// TIA Portal V20 export
DATA_BLOCK "Alarms"   // DB149
// stored: Access Published, MemoryReserve 100, Namespace Unit1
   VAR
      unitAlarms { ExternalWritable := 'False'} : "LAF_typeAlarms";
      emAlarms { ExternalWritable := 'False'} : Array[0.._.U1_NO_OF_EMs] of "LAF_typeAlarms";
      maintenanceFaults { ExternalWritable := 'False'} : Array[0..199] of Bool;   // PFE Maintenance Faults
      productionFaults { ExternalWritable := 'False'} : Array[0..199] of Bool;   // PFE Production Faults
      toolingFault { ExternalWritable := 'False'} : Array[0..199] of Bool;   // PFE Tooling Faults
      qualityFault { ExternalWritable := 'False'} : Array[0..199] of Bool;   // PFE Quality Faults
      throughputFaultBlocked { ExternalWritable := 'False'} : Array[0..199] of Bool;   // PFE Throughput Fault Blocked
      throughputFaultStarved { ExternalWritable := 'False'} : Array[0..199] of Bool;   // PFE Throughput Fault Starved
      throughputFault { ExternalWritable := 'False'} : Array[0..199] of Bool;   // PFE Throughput Fault
      systemFaultGeneral { ExternalWritable := 'False'} : Array[0..199] of Bool;   // PFE System Fault General
      materialFault { ExternalWritable := 'False'} : Array[0..199] of Bool;   // PFE Material Fault
      maintenanceWarnings { ExternalWritable := 'False'} : Array[0..199] of Bool;   // PFE Maintenance Warnings
      productionWarning { ExternalWritable := 'False'} : Array[0..199] of Bool;   // PFE Production Warning
      toolingWarning { ExternalWritable := 'False'} : Array[0..199] of Bool;   // PFE Tooling Warning
      qualityWarning { ExternalWritable := 'False'} : Array[0..199] of Bool;   // PFE Quality Warning
      throughputWarning { ExternalWritable := 'False'} : Array[0..199] of Bool;   // PFE Throughput Warning
      systemWarning { ExternalWritable := 'False'} : Array[0..199] of Bool;   // PFE System Warning
      materialWarning { ExternalWritable := 'False'} : Array[0..199] of Bool;   // PFE Material Warning
      maintenanceStatus { ExternalWritable := 'False'} : Array[0..199] of Bool;   // PFE Maintenance Status
      productionStatus { ExternalWritable := 'False'} : Array[0..199] of Bool;   // PFE Production Status
      toolingStatus { ExternalWritable := 'False'} : Array[0..199] of Bool;   // PFE Tooling Status
      qualityStatus { ExternalWritable := 'False'} : Array[0..199] of Bool;   // PFE Quality Status
      throughputStatus { ExternalWritable := 'False'} : Array[0..199] of Bool;   // PFE Throughput Status
      systemStatus { ExternalWritable := 'False'} : Array[0..199] of Bool;   // PFE System Status
      materialStatus { ExternalWritable := 'False'} : Array[0..199] of Bool;   // PFE Material Status
      tonMaintenanceFault { ExternalWritable := 'False'} : Array[0..199] of TON_TIME;   // PFE Maintenance Faults Ton Timer
      tonProductionFault { ExternalWritable := 'False'} : Array[0..199] of TON_TIME;   // PFE Production Faults Ton Timer
      tonToolingFault { ExternalWritable := 'False'} : Array[0..199] of TON_TIME;   // PFE Tooling Faults Ton Timer
      tonQualityFault { ExternalWritable := 'False'} : Array[0..199] of TON_TIME;   // PFE Quality Faults Ton Timer
      tonThroughputFaultBlocked { ExternalWritable := 'False'} : Array[0..199] of TON_TIME;   // PFE Throughput Fault Blocked Ton Timer
      tonThroughputFaultStarved { ExternalWritable := 'False'} : Array[0..199] of TON_TIME;   // PFE Throughput Fault Starved Ton Timer
      tonThroughputFault { ExternalWritable := 'False'} : Array[0..199] of TON_TIME;   // PFE Throughput Fault Ton Timer
      tonSystemFaultGeneral { ExternalWritable := 'False'} : Array[0..199] of TON_TIME;   // PFE System Fault General Ton Timer
      tonMaterialFault { ExternalWritable := 'False'} : Array[0..199] of TON_TIME;   // PFE Material Fault Ton Timer
      tonMaintenanceWarning { ExternalWritable := 'False'} : Array[0..199] of TON_TIME;   // PFE Maintenance Warnings Ton Timer
      tonProductionWarning { ExternalWritable := 'False'} : Array[0..199] of TON_TIME;   // PFE Production Warning Ton Timer
      tonToolingWarning { ExternalWritable := 'False'} : Array[0..199] of TON_TIME;   // PFE Tooling Warning Ton Timer
      tonQualityWarning { ExternalWritable := 'False'} : Array[0..199] of TON_TIME;   // PFE Quality Warning Ton Timer
      tonThroughputWarning { ExternalWritable := 'False'} : Array[0..199] of TON_TIME;   // PFE Throughput Warning Ton Timer
      tonSystemWarning { ExternalWritable := 'False'} : Array[0..199] of TON_TIME;   // PFE System Warning Ton Timer
      tonMaterialWarning { ExternalWritable := 'False'} : Array[0..199] of TON_TIME;   // PFE Material Warning Ton Timer
      tonMaintenanceStatus { ExternalWritable := 'False'} : Array[0..199] of TON_TIME;   // PFE Maintenance Status Ton Timer
      tonProductionStatus { ExternalWritable := 'False'} : Array[0..199] of TON_TIME;   // PFE Production Status Ton Timer
      tonToolingStatus { ExternalWritable := 'False'} : Array[0..199] of TON_TIME;   // PFE Tooling Status Ton Timer
      tonQualityStatus { ExternalWritable := 'False'} : Array[0..199] of TON_TIME;   // PFE Quality Status Ton Timer
      tonThroughputStatus { ExternalWritable := 'False'} : Array[0..199] of TON_TIME;   // PFE Throughput Status Ton Timer
      tonSystemStatus { ExternalWritable := 'False'} : Array[0..199] of TON_TIME;   // PFE System Status Ton Timer
      tonMaterialStatus { ExternalWritable := 'False'} : Array[0..199] of TON_TIME;   // PFE Material Status Ton Timer
      TonTimer { ExternalWritable := 'False'} : Array[0..99] of TON_TIME;
      NoDataTransfer { S7_SetPoint := 'True'} : Array[0..20] of Bool;
   END_VAR
BEGIN
   // maintenanceFaults[10] : OUT P&P GRIPPER 1ST Y-AXIS ROBOT HOME SENSOR
   // maintenanceFaults[11] : OUT P&P GRIPPER 2ND Y-AXIS ROBOT HOME SENSOR
   // maintenanceFaults[12] : OUT P&P GRIPPER 1ST Z-AXIS HOME SENSOR
   // maintenanceFaults[13] : OUT P&P GRIPPER 2ND Z-AXIS HOME SENSOR
   // maintenanceFaults[14] : TAPE Attachment ROBOT HOMING SENSOR
   // maintenanceFaults[15] : TOP TAPE fix STAGE ROBOT HOME SENSOR
   // maintenanceFaults[16] : SIDE TAPE Attachment FORWARD/BACKWARD ROBOT HOME SENSOR
   // maintenanceFaults[17] : SIDE TAPE Attachment MOVER ROBOT HOME SENSOR
   // maintenanceFaults[18] : SIDE TAPE FIX STAGE HOMING SENSOR
   // maintenanceFaults[19] : SIDE TAPE FIX STAGE ROTATION HOMING SENSOR
   // maintenanceFaults[20] : Thickness Z-AXIS HOME SENSOR
   // maintenanceFaults[21] : Process P&P X-axis Head#1 HOMING SENSOR
   // maintenanceFaults[22] : Process P&P X-axis Head#2 HOMING SENSOR
   // maintenanceFaults[23] : Process P&P Y-axis Head#1 HOMING SENSOR
   // maintenanceFaults[24] : Process P&P Z-axis Head#1 HOMING SENSOR
   // maintenanceFaults[25] : Process P&P Y-axis Head#2 HOMING SENSOR
   // maintenanceFaults[26] : Process P&P Z-axis Head#2 HOMING SENSOR
   // maintenanceFaults[27] : Unloading P&P X-axis HOMING SENSOR
   // maintenanceFaults[28] : Unloading P&P Z-axis HOMING SENSOR
   // maintenanceFaults[29] : Unloading P&P Θ-axis HOMING SENSOR
   // maintenanceFaults[30] : Brake Test After 24 Hours
   // systemFaultGeneral[0] : E202CB : KISTLER 100KN PRESS POWER TRIPPED
   // systemFaultGeneral[1] : E208CB : KISTLER 100KN PRESS POWER TRIPPED
   // systemFaultGeneral[2] : E214CB : KISTLER 30KN PRESS POWER TRIPPED
   // systemFaultGeneral[3] : SPARE
   // systemFaultGeneral[4] : SPARE
   // systemFaultGeneral[5] : E320CB : E8404PWS CONTROLLER POWER SMPS AC POWER TRIPPED
   // systemFaultGeneral[6] : E326CB : E8704PWS SAFETY POWER SMPS AC POWER TRIPPED
   // systemFaultGeneral[7] : E332CB : E8804PWS CONTRL POWER SMPS AC POWER TRIPPED
   // systemFaultGeneral[8] : E4120CB : PROCESSOR POWER ON TIPPRED
   // systemFaultGeneral[9] : E4126CB : PROGRAMING POWER OUTLET TRPPED
   // systemFaultGeneral[10] : SPARE
   // systemFaultGeneral[11] : E4304CB : PANEL LED POWER TRIPPED
   // systemFaultGeneral[12] : SPARE
   // systemFaultGeneral[13] : E4420CB : CONTROL LEVEL HUB POWER TRIPPED
   // systemFaultGeneral[14] : E4426CB : MAIN HMI POWER TRIPPED
   // systemFaultGeneral[15] : E4432CB : PORTABLE HMI POWER TIPPED
   // systemFaultGeneral[16] : E4456CB : PORTABLE HMI POWER TIPPED
   // systemFaultGeneral[17] : E5100CB : 120VAC HEATER-1 POWER TR PRIMARY TRIPPED
   // systemFaultGeneral[18] : SPARE
   // systemFaultGeneral[19] : SPARE
   // systemFaultGeneral[20] : E5156CB : UPPER 1-1 HEATER POWER TRIPPED
   // systemFaultGeneral[21] : E5162CB : UPPER 1-2 HEATER POWER TRIPPED
   // systemFaultGeneral[22] : E5168CB : LOWER 1-1 HEATER POWER TRIPPED
   // systemFaultGeneral[23] : E5174CB : LOWER 1-2 HEATER POWER TRIPPED
   // systemFaultGeneral[24] : E5180CB : LOWER 1-3 HEATER POWER TRIPPED
   // systemFaultGeneral[25] : SPARE
   // systemFaultGeneral[26] : E6100CB : 120VAC HEATER-2 POWER TR PRIMARY TRIPPED
   // systemFaultGeneral[27] : SPARE
   // systemFaultGeneral[28] : SPARE
   // systemFaultGeneral[29] : E6156CB : UPPER 2-1 HEATER POWER TRIPPED
   // systemFaultGeneral[30] : E6162CB : UPPER 2-2 HEATER POWER TRIPPED
   // systemFaultGeneral[31] : E6168CB : LOWER 2-1 HEATER POWER TRIPPED
   // systemFaultGeneral[32] : E6174CB : LOWER 2-2 HEATER POWER TRIPPED
   // systemFaultGeneral[33] : E6180CB : LOWER 2-3 HEATER POWER TRIPPED
   // systemFaultGeneral[34] : SPARE
   // systemFaultGeneral[35] : E7100CB : 120VAC CONTROL POWER TR PRIMARY TRIPPED
   // systemFaultGeneral[36] : E7110CB : 120VAC CONTROL POWER TR SECONDARY TRIPPED
   // systemFaultGeneral[37] : E7116CB : CONTROL POWER ON TRIPPED
   // systemFaultGeneral[38] : E7154CB : MOTOR PANEL CONTROL POWER TRIPPED
   // systemFaultGeneral[39] : E7160CB : POWER STRIP OUTLET POWER TRIPPED
   // systemFaultGeneral[40] : E7166CB : POWER STRIP OUTLET POWER TRIPPED
   // systemFaultGeneral[41] : E7172CB : QR LASER MARKING TRIPPED
   // systemFaultGeneral[42] : E7178CB : HI-POT TESTER POWER TRIPPED
   // systemFaultGeneral[43] : E7222CB : FFU-1 POWER TRIPPED
   // systemFaultGeneral[44] : E5206CB : UPPER 1-1 TEMPERATURE CONTROLLER POWER TRIPPED
   // systemFaultGeneral[45] : E5212CB : UPPER 1-2 TEMPERATURE CONTROLLER POWER TRIPPED
   // systemFaultGeneral[46] : E5218CB : LOWER 1-1 TEMPERATURE CONTROLLER POWER TRIPPED
   // systemFaultGeneral[47] : E5224CB : LOWER 1-2 TEMPERATURE CONTROLLER POWER TRIPPED
   // systemFaultGeneral[48] : E5230CB : LOWER 1-3 TEMPERATURE CONTROLLER POWER TRIPPED
   // systemFaultGeneral[49] : E6206CB : UPPER 2-1 TEMPERATURE CONTROLLER POWER TRIPPED
   // systemFaultGeneral[50] : E6212CB : UPPER 2-2 TEMPERATURE CONTROLLER POWER TRIPPED
   // systemFaultGeneral[51] : E6218CB : LOWER 2-1 TEMPERATURE CONTROLLER POWER TRIPPED
   // systemFaultGeneral[52] : E6224CB : LOWER 2-2 TEMPERATURE CONTROLLER POWER TRIPPED
   // systemFaultGeneral[53] : E6230CB : LOWER 2-3 TEMPERATURE CONTROLLER POWER TRIPPED
   // systemFaultGeneral[54] : SPARE
   // systemFaultGeneral[55] : E8154CB : ET200MP I/O OUTPUT POWER TRIPPED
   // systemFaultGeneral[56] : E8180CB : JUNCTION BOX CONTROL POWER TRIPPED
   // systemFaultGeneral[57] : E8204CB : CLASS 2 SMPS POWER TRIPPED
   // systemFaultGeneral[58] : E8220CB : ET200ECO PN-1 POWER TRIPPED
   // systemFaultGeneral[59] : E8224CB : ET200ECO PN-2 POWER TRIPPED
   // systemFaultGeneral[60] : E8228CB : ET200ECO PN-3 POWER TRIPPED
   // systemFaultGeneral[61] : E8232CB : ET200ECO PN-4 POWER TRIPPED
   // systemFaultGeneral[62] : E8304CB : PANEL FAN POWER TRIPPED
   // systemFaultGeneral[63] : SPARE
   // systemFaultGeneral[64] : E8406CB : CONTROLLER DC POWER TRIPPED
   // systemFaultGeneral[65] : E8416CB : KISTLER CONTROL POWER TRIPPED
   // systemFaultGeneral[66] : E8422CB : MANIFOLD-1 POWER TRIPPED
   // systemFaultGeneral[67] : E8430CB : MANIFOLD-2 POWER TRIPPED
   // systemFaultGeneral[68] : E8456CB : QR READER POWER TRIPPED
   // systemFaultGeneral[69] : E8462CB : QR READER POWER TRIPPED
   // systemFaultGeneral[70] : E8468CB : HANDY QR READER POWER TRIPPED
   // systemFaultGeneral[71] : E8474CB : PROFINET CONVERTER POWER TRIPPED
   // systemFaultGeneral[72] : E8504CB : MONITORING RELAY POWER TRIPPED
   // systemFaultGeneral[73] : SPARE
   // systemFaultGeneral[74] : E8706CB : SAFETY DC POWER TRIPPED
   // systemFaultGeneral[75] : E8716CB : ET200SP I/O SAFETY POWER TRIPPED
   // systemFaultGeneral[76] : E8736CB : JUNCTION BOX CONTROL POWER TRIPPED
   // systemFaultGeneral[77] : E8756CB : ET200ECO PN SAFETYT-1 POWER TRIPPED
   // systemFaultGeneral[78] : E8762CB : ET200ECO PN SAFETYT-2 POWER TRIPPED
   // systemFaultGeneral[79] : SPARE
   // systemFaultGeneral[80] : E8806CB : CONTROL DC POWER TRIPPED
   // systemFaultGeneral[81] : E8816CB : JUNCTION BOX CONTROL POWER TRIPPED
   // systemFaultGeneral[82] : E8822CB : DRIVE-CLIQ HUB POWER TRIPPED
   // systemFaultGeneral[83] : E8828CB : EQUIPMENT LED POWER TRIPPED
   // systemFaultGeneral[84] : E156CB : CONTROL DC POWER TRIPPED
   // systemFaultGeneral[85] : E218CB : SAFETY DC POWER TRIPPED
   // systemFaultGeneral[86] : E308CB : CLASS 2 SMPS POWER TRIPPED
   // systemFaultGeneral[87] : E324CB : ET200ECO PN-1 POWER TRIPPED
   // systemFaultGeneral[88] : E328CB : ET200ECO PN-2 POWER TRIPPED
   // systemFaultGeneral[89] : E332CB : ET200ECO PN-3 POWER TRIPPED
   // systemFaultGeneral[90] : E336CB : ET200ECO PN-4 POWER TRIPPED
   // systemFaultGeneral[91] : MOTOR POWER MC FEEDBACK
   // systemFaultGeneral[92] : E202CB : MOTOR POWER TRIPPED
   // systemFaultGeneral[93] : E208CB : MAIN CONTROL PANEL MAIN POWER TRIPPED
   // systemFaultGeneral[94] : E314CB : E6104PWS CONTROL POWER SMPS AC POWER TRIPPED
   // systemFaultGeneral[95] : E400CB : JROUT P&P Y-AXIS POWER TR PRIMARY TRIPPED
   // systemFaultGeneral[96] : E410CB : JROUT P&P Y-AXIS POWER TR ECONDARY TRIPPED
   // systemFaultGeneral[97] : E500CB : INS PROCESS P&P X-AXIS POWER TR PRIMARY TRIPPED
   // systemFaultGeneral[98] : E510CB : INS PROCESS P&P X-AXIS POWER TR ECONDARY TRIPPED
   // systemFaultGeneral[99] : E600CB : JR UNLOADING Y-AXIS POWER TR PRIMARY TRIPPED
   // systemFaultGeneral[100] : E610CB : JR UNLOADING Y-AXIS POWER TR ECONDARY TRIPPED
   // systemFaultGeneral[101] : E720CB : POWER METER POWER TRIIPED
   // systemFaultGeneral[102] : E726CB : POWER METER CONTROL POWER TRIIPED
   // systemFaultGeneral[103] : E2004CB : JR OUT P&P 1 Y-AXIS POWER ON TRIPPED
   // systemFaultGeneral[104] : E2104CB : JR OUT P&P 2 Y-AXIS POWER ON TRIPPED
   // systemFaultGeneral[105] : E2204CB : INS PROCESS P&P 1 X-AXIS POWER ON TRIPPED
   // systemFaultGeneral[106] : E2304CB : INS PROCESS P&P 2 X-AXIS POWER ON TRIPPED
   // systemFaultGeneral[107] : E2404CB : JR UNLOADING Y-AXIS POWER ON TRIPPED
   // systemFaultGeneral[108] : E6156CB : MOTOR POWER MC COIL POWER TRIPPED
   // systemFaultGeneral[109] : E4116CB : PROCESSOR POWER ON TRIPPRED
   // systemFaultGeneral[110] : E4156CB : MAIN CONTROL PANEL HOT POWER TRIPPED
   // systemFaultGeneral[111] : E4162CB : SYSTEM LEVEL HUB POWER TRIPPED
   // systemFaultGeneral[112] : E4304CB : PANEL LED POWER TRIPPED
   // systemFaultGeneral[113] : E5110CB : CONTROL POWER TRIPPED
   // systemFaultGeneral[114] : E5120CB : CONTROL POWER ON TRIPPED
   // systemFaultGeneral[115] : E6104PWS : CONTROL POWER SMPS DC
   // systemFaultGeneral[116] : E6122CB : SERVON CONTROL POWER TRIPPED
   // systemFaultGeneral[117] : E6128CB : SERVO CONTROL UNIT CONTROL POWER TRIPPED
   // systemFaultGeneral[118] : E6204CB : PANEL FAN POWER TRIPPED
   // systemFaultGeneral[119] : SPARE
   // systemFaultGeneral[120] : SPARE
   // systemFaultGeneral[121] : SPARE
   // systemFaultGeneral[122] : SPARE
   // systemFaultGeneral[123] : E4404PWS : PLC POWER SMPS DC
   // systemFaultGeneral[124] : E8104PWS : CONTROL POWER SMPS DC
   // systemFaultGeneral[125] : E8206PWS : CLASS 2 SMPS MONITORING
   // systemFaultGeneral[126] : E8404PWS : CONTROLLER POWER SMPS DC
   // systemFaultGeneral[127] : E8704PWS : SAFETY POWER SMPS DC
   // systemFaultGeneral[128] : E8804PWS : COONTRL POWER SMPS DC
   // systemFaultGeneral[129] : E310PWS : CLASS 2 SMPS MONITORING
   // systemFaultGeneral[130] : AIROK21 : MAIN AIR CLOSED
   // maintenanceWarnings[10] : 8 Hours Time Over
   // maintenanceWarnings[30] : Brake Test After 8 Hours
   // maintenanceWarnings[31] : Door unlock miss
   // NoDataTransfer[0] : Stack1 To JR Out P&P Left [BA030 → Em2]
   // NoDataTransfer[1] : Stack2 To JR Out P&P Left [BA040 → Em2]
   // NoDataTransfer[2] : JR Out P&P Left To Top Tape [Em2 → Em3]
   // NoDataTransfer[3] : Top Tape To JR Out P&P Right [Em3 → Em2]
   // NoDataTransfer[4] : JR Out P&P Right To Side Tape [Em2 → Em4]
   // NoDataTransfer[5] : Side Tape To Transfer P&P Left [Em4 → Em5]
   // NoDataTransfer[6] : Tr P&P Left To Hot Press Left [Em5 → Em6]
   // NoDataTransfer[7] : HotPress Left To Tr P&P Left [Em6 → Em5]
   // NoDataTransfer[8] : Tr P&P Left To HotPress Right [Em5 → Em7]
   // NoDataTransfer[9] : HotPress Right To Tr P&P Left [Em7 → Em5]
   // NoDataTransfer[10] : Tr P&P Left To Hipot & Thickness [Em5 → Em8]
   // NoDataTransfer[11] : Hipot Thickness To Tr P&P Right [Em8 → Em5]
   // NoDataTransfer[12] : Transfer P&P Right To Vision [Em5 → Em9]
   // NoDataTransfer[13] : Vision To Transfer P&P Right [Em9 → Em5]
   // NoDataTransfer[14] : Tr P&P Right To Laser Mark [Em5 → Em10]
   // NoDataTransfer[15] : Laser Mark To Tr P&P Right [Em10 → Em5]
   // NoDataTransfer[16] : Tr P&P Right To Weight Check [Em5 → Em11]
   // NoDataTransfer[17] : Weight Check To JR Unload P&P [Em11 → Em13]
END_DATA_BLOCK
